// TIA Portal V20 export
DATA_BLOCK "instAlarmCounter5"   // DB189
// stored: InstanceOfName LER_AlarmCounter_Sensor, InstanceOfType FB
"LER_AlarmCounter_Sensor"
   // VAR_INPUT
   //    productionMode : Bool;
   //    countUp : Bool;
   //    Sensor : Bool;
   //    detectTime : Time;
   // END_VAR
   // VAR_IN_OUT
   //    hmiInterface : "LER_typeAlarmCounterInterface";
   // END_VAR
   // VAR
   //    statPulse : Bool;
   //    statRisingEdge : Bool;
   //    statTonTimer : TON_TIME;
   //    statSensorOn : TON_TIME;
   //    statSensorOff : TON_TIME;
   // END_VAR
BEGIN
END_DATA_BLOCK
